// TIA Portal V20 export
// export: Created 2026-09-15T00:50:17.7541098Z, ExportSetting None, DisplayName Totally Integrated Automation Portal, DisplayVersion V20, DisplayName TIA Portal Openness, DisplayVersion V20, DisplayName TIA Portal Version Control Interface, DisplayVersion V20, DisplayName SINAMICS Startdrive Advanced, DisplayVersion V20, DisplayName SINAMICS Startdrive G130, G150, S120, S150, SINAMICS MV, G220, S200, S210, DisplayVersion V20, DisplayName SINAMICS Startdrive G110M, G120, G120C, G120D, G120P, G115D, DisplayVersion V20, DisplayName STEP 7 Professional, DisplayVersion V20, DisplayName STEP 7 Safety, DisplayVersion V20, DisplayName WinCC Basic/Comfort/Advanced, DisplayVersion V20, DisplayName WinCC Unified, DisplayVersion V20
FUNCTION_BLOCK "Graph_Sequencer"   // FB1, GRAPH
// stored: AutoNumber false, GraphVersion 6.0, InitialValuesAcquisition false, SetENOAutomatically false
   // inherited from GRAPH_BASE
   VAR_INPUT
      OFF_SQ { ExternalAccessible := 'False'; ExternalVisible := 'False'; ExternalWritable := 'False'} : Bool := false;   // 关闭顺控器
      INIT_SQ { ExternalAccessible := 'False'; ExternalVisible := 'False'; ExternalWritable := 'False'} : Bool := false;   // 将顺序设置为初始状态
      ACK_EF { ExternalAccessible := 'False'; ExternalVisible := 'False'; ExternalWritable := 'False'} : Bool := false;   // 确认所有的错误和故障
      S_PREV { ExternalAccessible := 'False'; ExternalVisible := 'False'; ExternalWritable := 'False'} : Bool := false;   // 在S_NO输出参数中显示前导步
      S_NEXT { ExternalAccessible := 'False'; ExternalVisible := 'False'; ExternalWritable := 'False'} : Bool := false;   // 在S_NO输出参数中显示后续步。
      SW_AUTO { ExternalAccessible := 'False'; ExternalVisible := 'False'; ExternalWritable := 'False'} : Bool := false;   // 自动模式
      SW_TAP { ExternalAccessible := 'False'; ExternalVisible := 'False'; ExternalWritable := 'False'} : Bool := false;   // 半自动/转换条件切换
      SW_TOP { ExternalAccessible := 'False'; ExternalVisible := 'False'; ExternalWritable := 'False'} : Bool := false;   // 半自动/忽略转换条件
      SW_MAN { ExternalAccessible := 'False'; ExternalVisible := 'False'; ExternalWritable := 'False'} : Bool := false;   // 手动模式
      S_SEL { ExternalAccessible := 'False'; ExternalVisible := 'False'; ExternalWritable := 'False'} : Int := 0;   // 选择要在 S_NO中输出的步。
      S_ON { ExternalAccessible := 'False'; ExternalVisible := 'False'; ExternalWritable := 'False'} : Bool := false;   // 激活S_NO 中显示的步。
      S_OFF { ExternalAccessible := 'False'; ExternalVisible := 'False'; ExternalWritable := 'False'} : Bool := false;   // 禁用 S_NO 中标识的步
      T_PUSH { ExternalAccessible := 'False'; ExternalVisible := 'False'; ExternalWritable := 'False'} : Bool := false;   // 允许在半自动模式下跳过转换条件。
   END_VAR
   VAR_OUTPUT
      S_NO { ExternalAccessible := 'False'; ExternalVisible := 'False'; ExternalWritable := 'False'} : Int := 0;   // 步编号
      S_MORE { ExternalAccessible := 'False'; ExternalVisible := 'False'; ExternalWritable := 'False'} : Bool := false;   // 更多步可用，并可在S_NO中显示。
      S_ACTIVE { ExternalAccessible := 'False'; ExternalVisible := 'False'; ExternalWritable := 'False'} : Bool := false;   // 在S_NO 中显示的步是激活的。
      ERR_FLT { ExternalAccessible := 'False'; ExternalVisible := 'False'; ExternalWritable := 'False'} : Bool := false;   // 互锁条件或监控条件组出错
      AUTO_ON { ExternalAccessible := 'False'; ExternalVisible := 'False'; ExternalWritable := 'False'} : Bool := false;   // 当前为自动模式
      TAP_ON { ExternalAccessible := 'False'; ExternalVisible := 'False'; ExternalWritable := 'False'} : Bool := false;   // 已启用SW_TAP模式。
      TOP_ON { ExternalAccessible := 'False'; ExternalVisible := 'False'; ExternalWritable := 'False'} : Bool := false;   // 启用半自动模式/忽略转换条件。
      MAN_ON { ExternalAccessible := 'False'; ExternalVisible := 'False'; ExternalWritable := 'False'} : Bool := false;   // 已启用手动模式。
   END_VAR
   VAR
      Trans43 { ExternalAccessible := 'False'; ExternalVisible := 'False'; ExternalWritable := 'False'; S7_SetPoint := 'True'} : G7_TransitionPlus_V6;
      Trans48 { ExternalAccessible := 'False'; ExternalVisible := 'False'; ExternalWritable := 'False'; S7_SetPoint := 'True'} : G7_TransitionPlus_V6;
      Trans49 { ExternalAccessible := 'False'; ExternalVisible := 'False'; ExternalWritable := 'False'; S7_SetPoint := 'True'} : G7_TransitionPlus_V6;
      Trans50 { ExternalAccessible := 'False'; ExternalVisible := 'False'; ExternalWritable := 'False'; S7_SetPoint := 'True'} : G7_TransitionPlus_V6;
      Trans51 { ExternalAccessible := 'False'; ExternalVisible := 'False'; ExternalWritable := 'False'; S7_SetPoint := 'True'} : G7_TransitionPlus_V6;
      Trans52 { ExternalAccessible := 'False'; ExternalVisible := 'False'; ExternalWritable := 'False'; S7_SetPoint := 'True'} : G7_TransitionPlus_V6;
      Trans55 { ExternalAccessible := 'False'; ExternalVisible := 'False'; ExternalWritable := 'False'; S7_SetPoint := 'True'} : G7_TransitionPlus_V6;
      Step30 { ExternalAccessible := 'False'; ExternalVisible := 'False'; ExternalWritable := 'False'; S7_SetPoint := 'True'} : G7_StepPlus_V6;
      Step31 { ExternalAccessible := 'False'; ExternalVisible := 'False'; ExternalWritable := 'False'; S7_SetPoint := 'True'} : G7_StepPlus_V6;
      Step32 { ExternalAccessible := 'False'; ExternalVisible := 'False'; ExternalWritable := 'False'; S7_SetPoint := 'True'} : G7_StepPlus_V6;
      Step33 { ExternalAccessible := 'False'; ExternalVisible := 'False'; ExternalWritable := 'False'; S7_SetPoint := 'True'} : G7_StepPlus_V6;
      Step34 { ExternalAccessible := 'False'; ExternalVisible := 'False'; ExternalWritable := 'False'; S7_SetPoint := 'True'} : G7_StepPlus_V6;
      Step36 { ExternalAccessible := 'False'; ExternalVisible := 'False'; ExternalWritable := 'False'; S7_SetPoint := 'True'} : G7_StepPlus_V6;
   END_VAR
BEGIN
// 顺序控制示例
// GRAPH 顺序控制示例
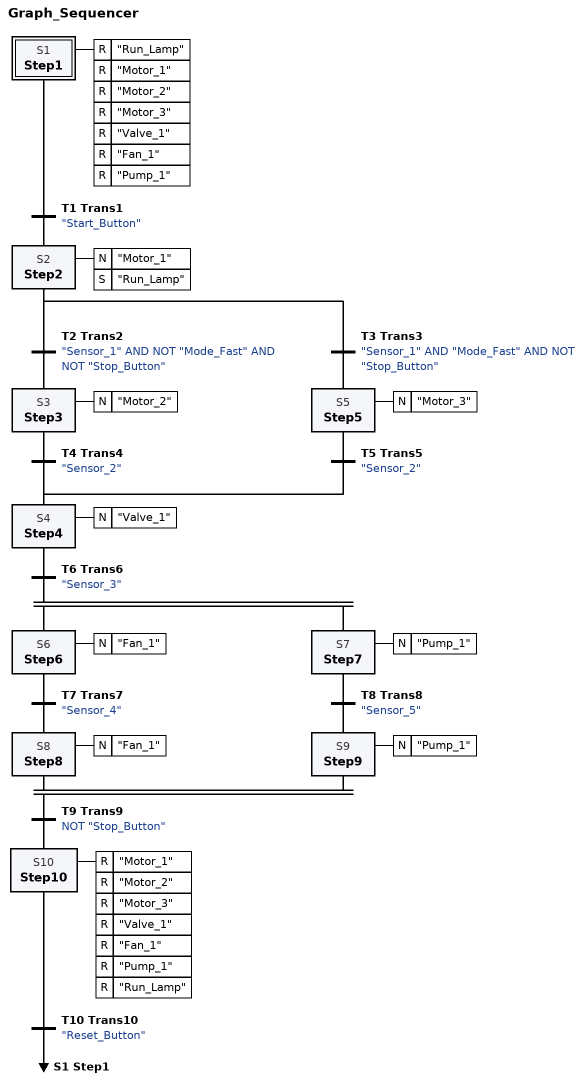
   // sequencer 1: 顺序控制示例：启动 → 送料 → 选择分支（正常/快速加工）→ 气缸 → 并行分支（冷却+润滑）→ 收尾 → 复位回初始步
   // GRAPH 顺序功能图示例（CPU 1511-1 PN）：含 1 个选择分支（AltBegin/AltEnd，按 Mode_Fast 二选一）与 1 个并行分支（SimBegin/SimEnd，冷却风机与润滑泵同时运行）。每步互锁 Interlock_Trip 为 1 时禁止本步动作，监控 Supervision_Trip 为 1 时触发监控故障。
   INITIAL_STEP Step1:   // S1, max time T#10S, warning time T#7S
      interlock C := NOT "Interlock_Trip";
      supervision V := "Supervision_Trip";
      // 初始步：等待启动
              R    "Run_Lamp"
              R    "Motor_1"
              R    "Motor_2"
              R    "Motor_3"
              R    "Valve_1"
              R    "Fan_1"
              R    "Pump_1"
   END_STEP
   TRANSITION Trans1 FROM Step1 TO Step2   // T1: 启动按钮 Start_Button
      := "Start_Button";
   END_TRANSITION
   STEP Step2:   // S2, max time T#10S, warning time T#7S
      interlock C := NOT "Interlock_Trip";
      supervision V := "Supervision_Trip";
      // 送料：电机 1 运行
              N    "Motor_1"
              S    "Run_Lamp"
   END_STEP
   TRANSITION Trans2 FROM Step2 TO Step3   // T2: 选择分支 A（正常模式）：送料到位 Sensor_1 且 非 Mode_Fast 且 未按停止
      := "Sensor_1" AND NOT "Mode_Fast" AND NOT "Stop_Button";
   END_TRANSITION
   TRANSITION Trans3 FROM Step2 TO Step5   // T3: 选择分支 B（快速模式）：送料到位 Sensor_1 且 Mode_Fast 且 未按停止
      := "Sensor_1" AND "Mode_Fast" AND NOT "Stop_Button";
   END_TRANSITION
   STEP Step3:   // S3, max time T#10S, warning time T#7S
      interlock C := NOT "Interlock_Trip";
      supervision V := "Supervision_Trip";
      // 选择分支 A：正常加工（电机 2 运行）
              N    "Motor_2"
   END_STEP
   TRANSITION Trans4 FROM Step3 TO Step4   // T4: 选择分支 A 加工完成 Sensor_2：进入汇合
      := "Sensor_2";
   END_TRANSITION
   STEP Step4:   // S4, max time T#10S, warning time T#7S
      interlock C := NOT "Interlock_Trip";
      supervision V := "Supervision_Trip";
      // 气缸推出
              N    "Valve_1"
   END_STEP
   TRANSITION Trans6 FROM Step4 TO (Step6, Step7)   // T6: 气缸到位 Sensor_3：进入并行分支
      := "Sensor_3";
   END_TRANSITION
   STEP Step5:   // S5, max time T#10S, warning time T#7S
      interlock C := NOT "Interlock_Trip";
      supervision V := "Supervision_Trip";
      // 选择分支 B：快速加工（电机 3 运行）
              N    "Motor_3"
   END_STEP
   TRANSITION Trans5 FROM Step5 TO Step4   // T5: 选择分支 B 加工完成 Sensor_2：进入汇合
      := "Sensor_2";
   END_TRANSITION
   STEP Step6:   // S6, max time T#10S, warning time T#7S
      interlock C := NOT "Interlock_Trip";
      supervision V := "Supervision_Trip";
      // 并行分支 A：冷却风机运行
              N    "Fan_1"
   END_STEP
   TRANSITION Trans7 FROM Step6 TO Step8   // T7: 并行分支 A：冷却到位 Sensor_4
      := "Sensor_4";
   END_TRANSITION
   STEP Step7:   // S7, max time T#10S, warning time T#7S
      interlock C := NOT "Interlock_Trip";
      supervision V := "Supervision_Trip";
      // 并行分支 B：润滑泵运行
              N    "Pump_1"
   END_STEP
   TRANSITION Trans8 FROM Step7 TO Step9   // T8: 并行分支 B：润滑到位 Sensor_5
      := "Sensor_5";
   END_TRANSITION
   STEP Step8:   // S8, max time T#10S, warning time T#7S
      interlock C := NOT "Interlock_Trip";
      supervision V := "Supervision_Trip";
      // 并行分支 A 结束步：保持冷却，等待汇合
              N    "Fan_1"
   END_STEP
   STEP Step9:   // S9, max time T#10S, warning time T#7S
      interlock C := NOT "Interlock_Trip";
      supervision V := "Supervision_Trip";
      // 并行分支 B 结束步：保持润滑，等待汇合
              N    "Pump_1"
   END_STEP
   TRANSITION Trans9 FROM (Step8, Step9) TO Step10   // T9: 两路并行全部完成 且 未按停止：进入收尾步
      := NOT "Stop_Button";
   END_TRANSITION
   STEP Step10:   // S10, max time T#10S, warning time T#7S
      interlock C := NOT "Interlock_Trip";
      supervision V := "Supervision_Trip";
      // 收尾：复位全部输出
              R    "Motor_1"
              R    "Motor_2"
              R    "Motor_3"
              R    "Valve_1"
              R    "Fan_1"
              R    "Pump_1"
              R    "Run_Lamp"
   END_STEP
   TRANSITION Trans10 FROM Step10 TO Step1   // T10, jump: 复位按钮回到初始步
      := "Reset_Button";
   END_TRANSITION
END_FUNCTION_BLOCK
